Staubli VAL3: TxtFile.dtx

public bool b7Axis
public bool b8Axis
public bool bActionWeldEnd[52]
public bool bAdjustSpEnable
public bool bAppro[6]
  [2] = true
  [3] = true
  [4] = true
  [5] = true
public bool bBypass[7]
public bool bLeave[2] = true
public bool bMatchPreset
public bool bMoreProd1Wp
public bool bMoveBack
public bool bMoveC[23]
public bool bOpenSharp
public bool bReadProduct
public bool bStartRead
public bool bSync7Axis
public bool bSync8Axis
public bool bTeachToolMode = true
public bool bTrajFilter
public bool bWeldEnable
public configRx cCfg
public frame fArray = {fatherId=fToffset[0]}
public frame fPofffset = {fatherId=fProduct[0]}
public frame fProduct = {x=-277.183, y=274.433, z=1513.292, rx=179.618, ry=-0.15, rz=0.135, fatherId=world[0]}
public frame fToffset = {fatherId=fTraj[0]}
public frame fTraj = {fatherId=fPofffset[0]}
public jointRx jAppro[6]
  [0] = {j1=37.473, j2=88.494, j3=-87.264, j4=-100.531, j5=89.054, j6=1.383}
  [1] = {j1=37.624, j2=77.945, j3=-75.448, j4=-100.7, j5=89.292, j6=2.626}
public jointRx jHome = {j1=33, j2=81, j3=-83, j4=-126, j5=90, j6=2}
public jointRx jLeave[2]
  [0] = {j1=34.791, j2=18.331, j3=101.066, j4=133.512, j5=-31.26, j6=40.017}
  [1] = {j1=38.12, j2=66.714, j3=-60.847, j4=-101.216, j5=89.968, j6=5.929}
mdesc mNomSpeed
mdesc mRun
public num nAction[51 12 2]
public num nExternalAxis[6]
num nFileBuffID
num nFileID
public num nHomeSpeed = 10
public num nMatchPreset[201 5]
public num nOpenShapeLeng
public num nPartTrajCount[100]
public num nPreset[51 5]
  [1,0] = 1
  [1,1] = 1
  [1,2] = 1
  [1,3] = 1
  [1,4] = 1
  [2,0] = 20
  [2,1] = 50
  [2,2] = 40
  [2,3] = 30
  [2,4] = 10
  [3,0] = 1
  [3,1] = 1
  [3,2] = 1
  [3,3] = 1
  [3,4] = 1
  [4,0] = 80
  [4,1] = 50
  [4,2] = 60
  [4,3] = 70
  [4,4] = 90
public num nReadCutCount
public num nReadTrajIndex = 1
public num nSingleType = 10
public num nStepLength
public num nTotalTraj = 7
public num nTrajDelay[2] = 0.3
public num nTrajIndex = 1
public num nTrajType[7]
  [0] = 10
  [1] = 10
  [2] = 10
  [3] = 10
  [4] = 10
  [5] = 10
  [6] = 9
public num nWeldActionId = 1.0863748
public pointRx pAppro[6]
  [0] = {fatherId=fArray[0]}
  [1] = {x=1202.964, y=578.195, z=257.373, rx=170.378, ry=1.129, rz=-130, fatherId=fArray[0]}
  [2] = {x=1200.953, y=-73.199, z=17.778, rx=178.998, ry=-0.002, rz=-62.905, fatherId=fArray[0]}
  [3] = {x=1200.953, y=-73.199, z=17.778, rx=178.998, ry=-0.002, rz=-62.905, fatherId=fArray[0]}
  [4] = {x=1200.953, y=-73.199, z=17.778, rx=178.998, ry=-0.002, rz=-62.905, fatherId=fArray[0]}
  [5] = {x=1200.953, y=-73.199, z=17.778, rx=178.998, ry=-0.002, rz=-62.905, fatherId=fArray[0]}
public pointRx pCut[23]
  [0] = {x=1200.196, y=-73.011, z=17.775, rx=178.998, ry=-0.002, rz=-62.905, fatherId=fArray[0]}
  [1] = {x=1199.424, y=-73.126, z=17.777, rx=178.998, ry=-0.002, rz=-62.905, fatherId=fArray[0]}
  [2] = {x=1198.755, y=-73.528, z=17.784, rx=178.998, ry=-0.002, rz=-62.905, fatherId=fArray[0]}
  [3] = {x=1198.291, y=-74.156, z=17.795, rx=178.998, ry=-0.002, rz=-62.905, fatherId=fArray[0]}
  [4] = {x=1197.953, y=-74.874, z=17.822, rx=178.998, ry=-0.002, rz=-62.905, fatherId=fArray[0]}
  [5] = {x=1197.758, y=-76.063, z=17.838, rx=178.998, ry=-0.002, rz=-62.905, fatherId=fArray[0]}
  [6] = {x=1198.207, y=-77.971, z=17.802, rx=178.998, ry=-0.002, rz=-62.905, fatherId=fArray[0]}
  [7] = {x=1199.208, y=-79.391, z=17.721, rx=178.998, ry=-0.002, rz=-62.905, fatherId=fArray[0]}
  [8] = {x=1200.754, y=-80.312, z=17.596, rx=178.998, ry=-0.002, rz=-62.905, fatherId=fArray[0]}
  [9] = {x=1202.535, y=-80.567, z=17.454, rx=178.998, ry=-0.002, rz=-62.905, fatherId=fArray[0]}
  [10] = {x=1204.293, y=-80.092, z=17.313, rx=178.998, ry=-0.002, rz=-62.905, fatherId=fArray[0]}
  [11] = {x=1205.733, y=-78.954, z=17.197, rx=178.998, ry=-0.002, rz=-62.905, fatherId=fArray[0]}
  [12] = {x=1206.543, y=-77.403, z=17.132, rx=178.998, ry=-0.002, rz=-62.905, fatherId=fArray[0]}
  [13] = {x=1206.76, y=-75.571, z=17.115, rx=178.998, ry=-0.002, rz=-62.905, fatherId=fArray[0]}
  [14] = {x=1206.253, y=-73.991, z=17.156, rx=178.998, ry=-0.002, rz=-62.905, fatherId=fArray[0]}
  [15] = {x=1205.134, y=-72.591, z=17.246, rx=178.998, ry=-0.002, rz=-62.905, fatherId=fArray[0]}
  [16] = {x=1203.479, y=-71.733, z=17.379, rx=178.998, ry=-0.002, rz=-62.905, fatherId=fArray[0]}
  [17] = {x=1201.681, y=-71.607, z=17.523, rx=178.998, ry=-0.002, rz=-62.905, fatherId=fArray[0]}
  [18] = {x=1199.977, y=-72.194, z=17.659, rx=178.998, ry=-0.002, rz=-62.905, fatherId=fArray[0]}
  [19] = {x=1198.665, y=-73.363, z=17.765, rx=178.998, ry=-0.002, rz=-62.905, fatherId=fArray[0]}
  [20] = {x=1197.953, y=-74.874, z=17.822, rx=178.998, ry=-0.002, rz=-62.905, fatherId=fArray[0]}
  [21] = {x=1197.758, y=-76.063, z=17.838, rx=178.998, ry=-0.002, rz=-62.905, fatherId=fArray[0]}
  [22] = {x=1198.207, y=-77.971, z=17.802, rx=178.998, ry=-0.002, rz=-62.905, fatherId=fArray[0]}
public pointRx pLeave[2]
  [0] = {x=1198.23, y=-78.003, z=17.8, rx=178.998, ry=-0.002, rz=-62.905, fatherId=fArray[0]}
  [1] = {fatherId=fArray[0]}
public pointRx pMoveC[23]
  [0] = {rx=-9.837, ry=-179.468, rz=-38.118, fatherId=fArray[0]}
  [1] = {fatherId=fArray[0]}
  [2] = {fatherId=fArray[0]}
  [3] = {fatherId=fArray[0]}
  [4] = {fatherId=fArray[0]}
  [5] = {fatherId=fArray[0]}
  [6] = {fatherId=fArray[0]}
  [7] = {fatherId=fArray[0]}
  [8] = {fatherId=fArray[0]}
  [9] = {fatherId=fArray[0]}
  [10] = {fatherId=fArray[0]}
  [11] = {fatherId=fArray[0]}
  [12] = {fatherId=fArray[0]}
  [13] = {fatherId=fArray[0]}
  [14] = {fatherId=fArray[0]}
  [15] = {fatherId=fArray[0]}
  [16] = {fatherId=fArray[0]}
  [17] = {fatherId=fArray[0]}
  [18] = {fatherId=fArray[0]}
  [19] = {fatherId=fArray[0]}
  [20] = {fatherId=fArray[0]}
  [21] = {fatherId=fArray[0]}
  [22] = {fatherId=fArray[0]}
public string sPresetName = "StaubliPreset"
public string sProductName = "123"
public string sTrajName[7]
  [0] = "123_1"
  [1] = "123_16"
  [2] = "123_17"
  [3] = "123_18"
  [4] = "123_19"
  [5] = "123_20"
  [6] = "123_23"
public string sTrajNameType[7]
  [0] = "123_1(不规则图形)"
  [1] = "123_16(不规则图形)"
  [2] = "123_17(不规则图形)"
  [3] = "123_18(不规则图形)"
  [4] = "123_19(不规则图形)"
  [5] = "123_20(不规则图形)"
  [6] = "123_23(同步空走路径)"
public string sTrajType[30]
  [1] = "圆-三点法(内切)"
  [2] = "圆-圆心直径(内切)"
  [3] = "三角形(内切)"
  [4] = "矩形(内切)"
  [5] = "正五边形(内切)"
  [6] = "正六边形(内切)"
  [7] = "腰形孔(内切)"
  [9] = "同步空走路径"
  [10] = "不规则图形"
  [11] = "圆-三点法(外切)"
  [12] = "圆-圆心直径(外切)"
  [13] = "三角形(外切)"
  [14] = "矩形(外切)"
  [15] = "正五边形(外切)"
  [16] = "正六边形(外切)"
  [17] = "腰形孔(外切)"
  [20] = "同步不规则图形"
  [21] = "五角星"
  [22] = "切圆管"
  [23] = "C形-圆心直径法"
  [24] = "C形-三点法"
public tool tCfg = {x=-239.363, y=-1.436, z=194.179, rx=-89.636, ry=-89.066, rz=-89.632, fatherId=flange[0]}
public tool tFileTool = {x=-239.363, y=-1.436, z=194.179, rx=-89.636, ry=-89.066, rz=-89.632, fatherId=flange[0]}
public trsf trAppro[6]
  [0] = {z=100, rx=5}
  [1] = {z=100, rx=5}
  [2] = {z=30, rx=80}
  [3] = {z=30, rx=80}
  [4] = {z=30, rx=80}
  [5] = {z=30, rx=80}
public trsf trApproAxis[6]
public trsf trArray
public trsf trAxis8Data = {y=0.001, z=1, rx=1}
public trsf trAxisData = {y=0.001, z=1, rx=1}
public trsf trBoxcar
public trsf trCorner = {x=1, z=100, rx=15, ry=5}
public trsf trCut[23]
  [0] = {z=30, rx=80}
  [1] = {x=1, z=30, rx=80}
  [2] = {x=1, z=30, rx=80}
  [3] = {z=30, rx=80}
  [4] = {x=1, z=30, rx=80}
  [5] = {x=1, z=30, rx=80}
  [6] = {x=1, z=30, rx=80}
  [7] = {x=1, z=30, rx=80}
  [8] = {x=1, z=30, rx=80}
  [9] = {x=1, z=30, rx=80}
  [10] = {x=1, z=30, rx=80}
  [11] = {x=1, z=30, rx=80}
  [12] = {x=1, z=30, rx=80}
  [13] = {x=1, z=30, rx=80}
  [14] = {x=1, z=30, rx=80}
  [15] = {x=1, z=30, rx=80}
  [16] = {x=1, z=30, rx=80}
  [17] = {x=1, z=30, rx=80}
  [18] = {x=1, z=30, rx=80}
  [19] = {x=1, z=30, rx=80}
  [20] = {x=1, z=30, rx=80}
  [21] = {x=1, z=30, rx=80}
  [22] = {x=1, z=30, rx=80}
public trsf trCutAxis[23]
public trsf trDefaultFrame
public trsf trDownLead = {ry=8}
public trsf trIODelay = {x=0.2, y=0.2}
public trsf trLeave[2]
  [0] = {z=30, rx=80}
  [1] = {z=100, rx=5}
public trsf trLeaveAxis[2]
public trsf trPointCount = {x=6, y=23, z=2}
public trsf trPresetData = {x=2000, y=200, z=32700}
public trsf trReguPara[3]
  [0] = {x=1, z=25, rx=1, ry=0.05}
  [1] = {x=1, z=25, rx=1, ry=0.05}
  [2] = {x=1, z=25, rx=1, ry=0.05}
public trsf trRegular[3]
  [0] = {x=1205.647, y=700.52, z=95.638, rx=-9.837, ry=-179.468, rz=-38.118}
  [1] = {x=1204.5, y=694.721, z=96.662, rx=-9.837, ry=-179.468, rz=-38.118}
  [2] = {x=1192.5, y=694.721, z=96.662, rx=-9.838, ry=-179.468, rz=-38.118}
public trsf trSync7Axis
public trsf trSync8Axis
public trsf trWorkplace = {x=11507, y=50, z=11507, rx=50, rz=-1}
